{attribute 'pack_mode' := '2'}
TYPE ST_LIST_STATE :
STRUCT
  Init        : E_PROGRESS;
  State       : E_LIST_STATE;

  Free        : UDINT;
  Count       : UDINT;
END_STRUCT
END_TYPE

(* stored: Version 1.1.0.1, ProductVersion 3.1.4026.18
   DUT ST_LIST_STATE: Id {c8554b59-d176-4eb1-804f-0c5b038cdcf0} *)
